{attribute 'Tc2GvlVarNames'}
VAR_CONFIG
END_VAR

(* stored: Version 1.1.0.1, ProductVersion 3.1.4024.0
   GVL Variable_Configuration: Id {4a21b063-0d92-458f-a316-0a38f8cef5d9} *)
